FUNCTION_BLOCK FB_WriteLog
VAR_IN_OUT
	bWrite:BOOL;
END_VAR
VAR_INPUT	
	sFileName:STRING;
	sMessage : STRING;
END_VAR

VAR_OUTPUT
	OK:BOOL;
	Busy:BOOL;
	ErrorMsg:STRING(255);
	bError:BOOL;
	ErrorID:UDINT;
END_VAR

VAR
	fileOpen:FB_FileOpen;
	fileWrite:FB_FileWrite;
	fileClose:FB_FileClose;
	fileDelete:FB_FileDelete;
	hFile:UINT;
	stringBuffer:STRING(255);
	eWriteStep:INT;
	sFileExtendName:STRING(255);
	LengthOfFileName:INT;
	
	iArrNo:UINT;
	rtWriteCSV:R_trig;
	bReset: BOOL;
	GetTimeStartDelay: Ton;
	NT_GetTime1: NT_GetTime;
	TIMESTR1: TIMESTRUCT;
	sCurrentTime_Temp: STRING;
END_VAR

NT();

rtWriteCSV(CLK:=bWrite,Q=>);

CASE eWriteStep OF
0:
	Busy:=FALSE;
	IF bWrite   THEN
		bWrite := FALSE;
		OK:=FALSE;
		Busy:=TRUE;
		iArrNo:=0;
		bError:=FALSE;
		ErrorMsg:='';
		ErrorID:=0;
		eWriteStep:=100;	
	END_IF
	
(*判断文件扩展名是否正确*)	
100:	
	fileOpen(bExecute:=TRUE);
	IF fileOpen.bBusy THEN
		eWriteStep:=210;	
	END_IF

210:
	fileOpen(bExecute:=FALSE);
	IF NOT fileOpen.bBusy AND NOT fileOpen.bError THEN
		eWriteStep:=300;	
	END_IF
	IF fileOpen.bError THEN
		ErrorMsg:='FileOpenError';
		ErrorID:=fileOpen.nErrId;
		eWriteStep:=9999;	
	END_IF

300:
		stringBuffer:='';
		stringBuffer:=CONCAT(stringBuffer,sCurrentTime_Temp);
		stringBuffer:=CONCAT(stringBuffer,'->');
		stringBuffer:=CONCAT(stringBuffer,sMessage);
		stringBuffer:=CONCAT(stringBuffer,'$n');
		fileWrite(bExecute:=TRUE,cbWriteLen:=LEN(stringBuffer));
		IF fileWrite.bBusy THEN
			eWriteStep:=310;	
		END_IF
310:
	fileWrite(bExecute:=FALSE);
	IF NOT fileWrite.bBusy AND NOT fileWrite.bError THEN
		eWriteStep:=500;	
	END_IF
	IF fileWrite.bError THEN
		ErrorMsg:='FileWriteError';
		ErrorID:=fileWrite.nErrId;
		eWriteStep:=9999;	
	END_IF

500:
	fileClose(bExecute:=TRUE);
	IF fileClose.bBusy THEN
		eWriteStep:=510;	
	END_IF

510:
	fileClose(bExecute:=FALSE);
	IF NOT fileClose.bBusy AND NOT fileClose.bError THEN
		eWriteStep:=600;	
	END_IF
	IF fileClose.bError THEN
		ErrorMsg:='FileOpenError';
		ErrorID:=fileOpen.nErrId;
		eWriteStep:=9999;	
	END_IF
	
600:
	OK:=TRUE;
	eWriteStep:=0;	
		
9999:
	bError:=TRUE;
	Busy:=FALSE;
	IF bReset THEN
		OK:=FALSE;
		ErrorID:=0;
		eWriteStep:=0;	
	END_IF
	
END_CASE

Act01_CallFB();

ACTION Act01_CallFB:
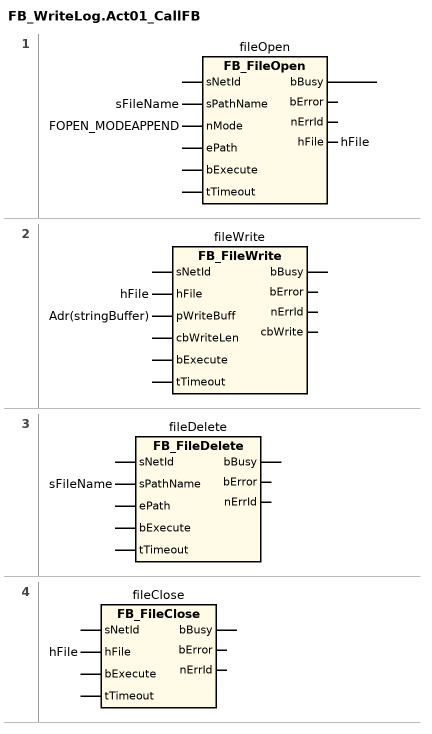
// NETWORK 1
fileOpen(sPathName := sFileName, nMode := FOPEN_MODEAPPEND, hFile => hFile); // FB_FileOpen

// NETWORK 2
fileWrite(hFile := hFile, pWriteBuff := Adr(stringBuffer)); // FB_FileWrite

// NETWORK 3
fileDelete(sPathName := sFileName); // FB_FileDelete

// NETWORK 4
fileClose(hFile := hFile); // FB_FileClose
END_ACTION

ACTION NT:

GetTimeStartDelay(IN:=NOT GetTimeStartDelay.Q  , PT:=T#1S , Q=> , ET=> );
NT_GetTime1(
	NETID:= ,
	START:=GetTimeStartDelay.Q ,
	TMOUT:= , 
	BUSY=> ,
	ERR=> ,
	ERRID=> ,
	TIMESTR=>TIMESTR1 );

TIMESTR1.wYear;		(*年*)
TIMESTR1.wMonth;		(*月*)
TIMESTR1.wDay;		(*日*)
TIMESTR1.wHour;		(*时*)
TIMESTR1.wMinute;		(*分*)
TIMESTR1.wSecond;		(*秒*)
TIMESTR1.wMilliseconds;	(*毫秒*)
TIMESTR1.wDayOfWeek;	(*星期*)

sCurrentTime_Temp := '';
sCurrentTime_Temp := CONCAT(sCurrentTime_Temp,WORD_TO_STRING(TIMESTR1.wYear));
 sCurrentTime_Temp:= CONCAT(sCurrentTime_Temp,'-');
 sCurrentTime_Temp:= CONCAT(sCurrentTime_Temp,WORD_TO_STRING(TIMESTR1.wMonth));
 sCurrentTime_Temp:= CONCAT(sCurrentTime_Temp,'-');
 sCurrentTime_Temp:= CONCAT(sCurrentTime_Temp,WORD_TO_STRING(TIMESTR1.wDay));
 sCurrentTime_Temp:= CONCAT(sCurrentTime_Temp,' ');
 sCurrentTime_Temp:= CONCAT(sCurrentTime_Temp,WORD_TO_STRING(TIMESTR1.wHour));
sCurrentTime_Temp := CONCAT(sCurrentTime_Temp,':');
 sCurrentTime_Temp:= CONCAT(sCurrentTime_Temp,WORD_TO_STRING(TIMESTR1.wMinute));
 sCurrentTime_Temp:= CONCAT(sCurrentTime_Temp,':');
 sCurrentTime_Temp:= CONCAT(sCurrentTime_Temp,WORD_TO_STRING(TIMESTR1.wSecond));
END_ACTION

END_FUNCTION_BLOCK

(* stored: Version 1.1.0.1, ProductVersion 3.1.4024.12
   POU FB_WriteLog: Id {22896bc6-5e49-4c45-8372-5786ffe05552}, SpecialFunc None
   Action Act01_CallFB: Id {55168cff-5397-4d02-a066-31f2563a9987}
   Action NT: Id {e6e039c3-b261-4141-9510-d89e6dc74d24} *)
